FUNCTION_BLOCK PUBLIC RestorePreviousAutomaticState
VAR_INPUT
END_VAR
VAR_OUTPUT
END_VAR
VAR
	RotationRestored: BOOL := FALSE;
	LiftingRestored: BOOL := FALSE;
	ExtensionRestored: BOOL := FALSE;
	GripRestored: BOOL := FALSE;
END_VAR

IF IO.PreviousManualMode THEN
	Automatic.AllRestored := FALSE;
END_IF

// reset rotation:
IF Automatic.RotationPositionAuto - Automatic.RotationPositionCurrent > 5 AND (NOT RotationRestored) AND (NOT Automatic.SafetyRON) THEN
	IO.MotorRotationDirection := 0;
	Automatic.RCurrentlyMoving := TRUE;
	IO.MotorRotation := 1;
ELSIF Automatic.RotationPositionCurrent - Automatic.RotationPositionAuto > 5 AND (NOT RotationRestored) AND (NOT Automatic.SafetyRON) THEN
	IO.MotorRotationDirection := 1;
	Automatic.RCurrentlyMoving := TRUE;
	IO.MotorRotation := 1;
ELSE
	Automatic.RCurrentlyMoving := FALSE;
	IO.MotorRotation := 0;
	RotationRestored := TRUE;
END_IF

// reset lifting:
IF Automatic.LiftingPositionAuto - Automatic.LiftingPositionCurrent > 5 AND (NOT LiftingRestored) AND (NOT Automatic.SafetyLON) THEN
	IO.MotorLiftingDirection := 0;
	Automatic.LCurrentlyMoving := TRUE;
	IO.MotorLifting := 1;
ELSIF Automatic.LiftingPositionCurrent - Automatic.LiftingPositionAuto > 5 AND (NOT LiftingRestored) AND (NOT Automatic.SafetyLON) THEN
	IO.MotorLiftingDirection := 0;
	Automatic.LCurrentlyMoving := TRUE;
	IO.MotorLifting := 1;
ELSE
	Automatic.LCurrentlyMoving := FALSE;
	IO.MotorLifting := 0;
	LiftingRestored := TRUE;
END_IF

// reset extension:
IF Automatic.ExtensionPositionAuto - Automatic.ExtensionPositionCurrent > 5 AND (NOT ExtensionRestored) AND (NOT Automatic.SafetyEON) THEN
	IO.MotorExtensionDirection := 0;
	Automatic.ECurrentlyMoving := TRUE;
	IO.MotorExtension := 1;
ELSIF Automatic.ExtensionPositionCurrent - Automatic.ExtensionPositionAuto > 5 AND (NOT ExtensionRestored) AND (NOT Automatic.SafetyEON) THEN
	IO.MotorExtensionDirection := 0;
	Automatic.ECurrentlyMoving := TRUE;
	IO.MotorExtension := 1;
ELSE
	Automatic.ECurrentlyMoving := FALSE;
	IO.MotorExtension := 0;
	ExtensionRestored := TRUE;
END_IF

// reset grip:
IF Automatic.GripPositionAuto - Automatic.GripPositionCurrent > 5 AND (NOT GripRestored) AND (NOT Automatic.SafetyGON) THEN
	IO.MotorGripDirection := 0;
	Automatic.GCurrentlyMoving := TRUE;
	IO.MotorGrip := 1;
ELSIF Automatic.GripPositionCurrent - Automatic.GripPositionAuto > 5 AND (NOT GripRestored) AND (NOT Automatic.SafetyGON) THEN
	IO.MotorGripDirection := 0;
	Automatic.GCurrentlyMoving := TRUE;
	IO.MotorGrip := 1;
ELSE
	Automatic.GCurrentlyMoving := FALSE;
	IO.MotorGrip := 0;
	GripRestored := TRUE;
END_IF

// if all restored then go on to exeecute recipes in AutomaticControl:
IF RotationRestored AND LiftingRestored AND ExtensionRestored AND GripRestored THEN
	IO.PreviousManualMode := FALSE;
	Automatic.AllRestored := TRUE;
	
	RotationRestored := FALSE;
	ExtensionRestored := FALSE;
	LiftingRestored := FALSE;
	GripRestored := FALSE;
	Automatic.RCurrentlyMoving := FALSE;
	Automatic.ECurrentlyMoving := FALSE;
	Automatic.LCurrentlyMoving := FALSE;
	Automatic.GCurrentlyMoving := FALSE;
END_IF

END_FUNCTION_BLOCK

(* stored: Version 1.1.0.1, ProductVersion 3.1.4024.13
   POU RestorePreviousAutomaticState: Id {bf2e792f-bc3c-4ce2-afd6-05125fa35279}, SpecialFunc None *)
